{attribute 'qualified_only'}
VAR_GLOBAL
	P1 AT %Q*:BOOL; 	// Meldeleuchte weiss
	P2 AT %Q*:BOOL;     // Meldeleuchte grün
	P3 AT %Q*:BOOL;		// Meldeleuchte rot
	Q1 AT %Q*:BOOL;     // Motor Schnell (RL)
	Q2 AT %Q*:BOOL;     // Motor Linkslauf
	Q3 AT %Q*:BOOL;     // Motor Langsam (RL)
END_VAR

(* stored: Version 1.1.0.1, ProductVersion 3.1.4024.5
   GVL DA: Id {efa3d63a-96e1-4204-b1e7-9f3703bd4f03} *)
